(* IEC 61131-3 sources: mect_apps/TPAC1007_04_AA/Octopus_Prey_PLC, 1 file *)

(* ---- Program1.st ---- *)
(*[[
]]*)
PROGRAM Program1
#import "Crosstable.gvl"
VAR
	first : bool := true;
END_VAR
	(* Initial Configuration *)
	if first then
 	    first := false;
		PLC_DigDir_1 := 0; (* input *)
		PLC_DigDir_2 := 0; (* input *)
		PLC_DigDir_3 := 0; (* input *)
		PLC_DigDir_4 := 0; (* input *)
		PLC_DigDir_5 := 0; (* input *)
		PLC_DigDir_6 := 0; (* input *)
		PLC_DigDir_7 := 0; (* input *)
		PLC_DigDir_8 := 0; (* input *)
		PLC_AnInConf_1 := 2; (* 0..10V *)
		PLC_AnInConf_2 := 2; (* 0..10V *)
		PLC_AnOutConf_1 := 2; (* 0..10V *)
		PLC_AnOutConf_2 := 2; (* 0..10V *)
		PLC_AnOutConf_3 := 2; (* 0..10V *)
		PLC_AnOutConf_4 := 2; (* 0..10V *)
	end_if;
END_PROGRAM
